(* PLC project Tc2_Utilities.PLC_ReadSymInfo Demo, tc3-libraries-kb TwinCAT 3.1 *)
(* stored: creationDateTime 2026-05-10T20:00:00, modificationDateTime 2026-05-10T20:00:00 *)

PROGRAM P_Demo_PLC_ReadSymInfo
  VAR
    fbPLC_ReadSymInfo : PLC_ReadSymInfo;  (* Tc2_Utilities.PLC_ReadSymInfo 实例 *)
    arg_NETID : T_AmsNetId;  (* VAR_INPUT NETID *)
    arg_PORT : T_AmsPort;  (* VAR_INPUT PORT *)
    arg_START : BOOL;  (* VAR_INPUT START *)
    arg_TMOUT : TIME;  (* VAR_INPUT TMOUT *)
    out_BUSY : BOOL;  (* VAR_OUTPUT BUSY *)
    out_ERR : BOOL;  (* VAR_OUTPUT ERR *)
    out_ERRID : UDINT;  (* VAR_OUTPUT ERRID *)
    out_SYMCOUNT : UDINT;  (* VAR_OUTPUT SYMCOUNT *)
    out_SYMSIZE : UDINT;  (* VAR_OUTPUT SYMSIZE *)
  END_VAR

            // ============================================================
// Tc2_Utilities.PLC_ReadSymInfo 演示程序（FB 实例）
// ============================================================
// 验证步骤：
//   1. 引用 Tc2_Utilities（及依赖类型所在库 Tc2_System 等）
//   2. 编译 + 登录
//   3. 按 doc.md 给 arg_* 赋值
//   4. 在线监视 out_* / io_* 输出
// ============================================================

fbPLC_ReadSymInfo(
    NETID := arg_NETID,
    PORT := arg_PORT,
    START := arg_START,
    TMOUT := arg_TMOUT,
    BUSY => out_BUSY,
    ERR => out_ERR,
    ERRID => out_ERRID,
    SYMCOUNT => out_SYMCOUNT,
    SYMSIZE => out_SYMSIZE
);

          
END_PROGRAM
